FUNCTION_BLOCK HHM_FV_PART_1
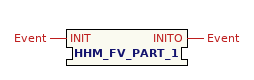
  EVENT_INPUT
    INIT;
  END_EVENT
  EVENT_OUTPUT
    INITO;
  END_EVENT
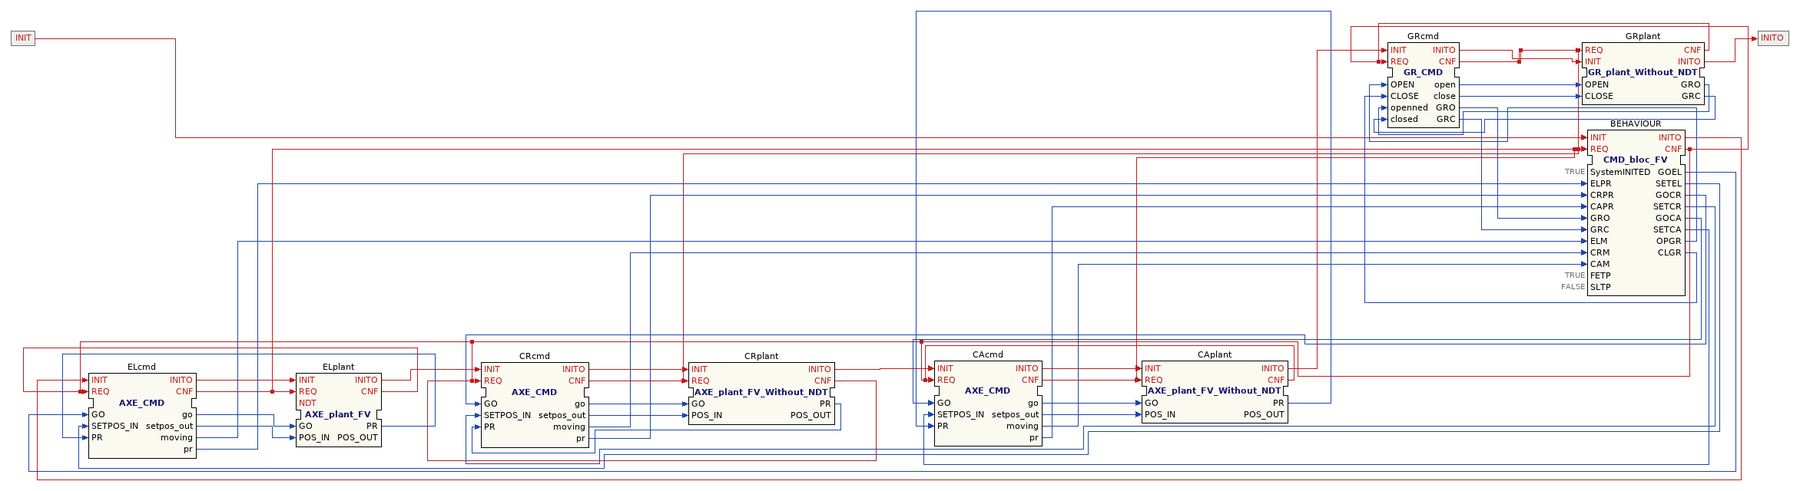
  FBS
    ELcmd : AXE_CMD;
    ELplant : AXE_plant_FV;
    CRcmd : AXE_CMD;
    CRplant : AXE_plant_FV_Without_NDT;
    CAcmd : AXE_CMD;
    CAplant : AXE_plant_FV_Without_NDT;
    GRplant : GR_plant_Without_NDT;
    GRcmd : GR_CMD;
    BEHAVIOUR : CMD_bloc_FV(FETP := TRUE, SLTP := FALSE, SystemINITED := TRUE);
  END_FBS
  EVENT_CONNECTIONS
    ELcmd.INITO TO ELplant.INIT;
    ELcmd.CNF TO ELplant.REQ;
    CRcmd.INITO TO CRplant.INIT;
    CRcmd.CNF TO CRplant.REQ;
    CRplant.CNF TO CRcmd.REQ;
    CAcmd.INITO TO CAplant.INIT;
    CAcmd.CNF TO CAplant.REQ;
    CAplant.CNF TO CAcmd.REQ;
    ELplant.CNF TO ELcmd.REQ;
    GRcmd.CNF TO GRplant.REQ;
    GRcmd.INITO TO GRplant.INIT;
    BEHAVIOUR.CNF TO ELcmd.REQ;
    BEHAVIOUR.CNF TO CRcmd.REQ;
    ELcmd.CNF TO BEHAVIOUR.REQ;
    CRcmd.CNF TO BEHAVIOUR.REQ;
    BEHAVIOUR.CNF TO CAcmd.REQ;
    CAcmd.CNF TO BEHAVIOUR.REQ;
    BEHAVIOUR.CNF TO GRcmd.REQ;
    BEHAVIOUR.INITO TO ELcmd.INIT;
    ELplant.INITO TO CRcmd.INIT;
    CRplant.INITO TO CAcmd.INIT;
    CAplant.INITO TO GRcmd.INIT;
    GRplant.CNF TO GRcmd.REQ;
    GRcmd.CNF TO BEHAVIOUR.REQ;
    INIT TO BEHAVIOUR.INIT;
    GRplant.INITO TO INITO;
  END_CONNECTIONS
  DATA_CONNECTIONS
    ELcmd.go TO ELplant.GO;
    ELplant.PR TO ELcmd.PR;
    CRcmd.go TO CRplant.GO;
    CRplant.PR TO CRcmd.PR;
    CAcmd.go TO CAplant.GO;
    CAplant.PR TO CAcmd.PR;
    GRcmd.open TO GRplant.OPEN;
    GRcmd.close TO GRplant.CLOSE;
    GRplant.GRO TO GRcmd.openned;
    GRplant.GRC TO GRcmd.closed;
    BEHAVIOUR.GOEL TO ELcmd.GO;
    BEHAVIOUR.SETEL TO ELcmd.SETPOS_IN;
    ELcmd.moving TO BEHAVIOUR.ELM;
    ELcmd.pr TO BEHAVIOUR.ELPR;
    BEHAVIOUR.GOCR TO CRcmd.GO;
    BEHAVIOUR.SETCR TO CRcmd.SETPOS_IN;
    CRcmd.pr TO BEHAVIOUR.CRPR;
    CAcmd.pr TO BEHAVIOUR.CAPR;
    BEHAVIOUR.GOCA TO CAcmd.GO;
    BEHAVIOUR.SETCA TO CAcmd.SETPOS_IN;
    BEHAVIOUR.OPGR TO GRcmd.OPEN;
    BEHAVIOUR.CLGR TO GRcmd.CLOSE;
    GRcmd.GRO TO BEHAVIOUR.GRO;
    GRcmd.GRC TO BEHAVIOUR.GRC;
    CRcmd.moving TO BEHAVIOUR.CRM;
    CAcmd.moving TO BEHAVIOUR.CAM;
    ELcmd.setpos_out TO ELplant.POS_IN;
    CRcmd.setpos_out TO CRplant.POS_IN;
    CAcmd.setpos_out TO CAplant.POS_IN;
  END_CONNECTIONS
END_FUNCTION_BLOCK
